LIN {X 0,Y 117.443,Z 618.499,A -85,B 0,C 180,E1 -30787.751,E2 -30787.751} C_VEL
LIN {X 0,Y 117.759,Z 615.991,A -85,B 0,C 180,E1 -30784.552,E2 -30784.552} C_VEL
LIN {X 0,Y 118.169,Z 614.006,A -85,B 0,C 180,E1 -30779.995,E2 -30779.995} C_VEL
LIN {X 0,Y 117.877,Z 614.864,A -85,B 0,C 180,E1 -30779.723,E2 -30779.723} C_VEL
LIN {X 0,Y 113.586,Z 625.245,A -85,B 0,C 180,E1 -30779.502,E2 -30779.502} C_VEL
LIN {X 0,Y 107.189,Z 637.349,A -85,B 0,C 180,E1 -30779.105,E2 -30779.105} C_VEL
LIN {X 0,Y 99.299,Z 648.745,A -85,B 0,C 180,E1 -30778.609,E2 -30778.609} C_VEL
LIN {X 0,Y 93.168,Z 656.16,A -85,B 0,C 180,E1 -30778.155,E2 -30778.155} C_VEL
LIN {X 0,Y 84.423,Z 664.947,A -85,B 0,C 180,E1 -30777.39,E2 -30777.39} C_VEL
LIN {X 0,Y 77.444,Z 670.933,A -85,B 0,C 180,E1 -30776.591,E2 -30776.591} C_VEL
LIN {X 0,Y 68.748,Z 677.241,A -85,B 0,C 180,E1 -30775.357,E2 -30775.357} C_VEL
LIN {X 0,Y 59.764,Z 682.696,A -85,B 0,C 180,E1 -30773.548,E2 -30773.548} C_VEL
LIN {X 0,Y 49.831,Z 687.613,A -85,B 0,C 180,E1 -30770.836,E2 -30770.836} C_VEL
LIN {X 0,Y 39.702,Z 691.58,A -85,B 0,C 180,E1 -30766.802,E2 -30766.802} C_VEL
LIN {X 0,Y 29.884,Z 694.52,A -85,B 0,C 180,E1 -30760.167,E2 -30760.167} C_VEL
LIN {X 0,Y 23.763,Z 696.03,A -85,B 0,C 180,E1 -30752.531,E2 -30752.531} C_VEL
LIN {X 0,Y 14.258,Z 697.578,A -85,B 0,C 180,E1 -30719.533,E2 -30719.533} C_VEL
LIN {X 0,Y 12.869,Z 697.867,A -85,B 0,C 180,E1 -30690,E2 -30690} C_VEL
LIN {X 0,Y 18.308,Z 696.97,A -85,B 0,C 180,E1 -30639.849,E2 -30639.849} C_VEL
LIN {X 0,Y 23.763,Z 696.03,A -85,B 0,C 180,E1 -30627.469,E2 -30627.469} C_VEL
LIN {X 0,Y 36.383,Z 692.67,A -85,B 0,C 180,E1 -30615.024,E2 -30615.024} C_VEL
LIN {X 0,Y 46.428,Z 689.041,A -85,B 0,C 180,E1 -30610.286,E2 -30610.286} C_VEL
LIN {X 0,Y 56.667,Z 684.307,A -85,B 0,C 180,E1 -30607.176,E2 -30607.176} C_VEL
LIN {X 0,Y 65.281,Z 679.425,A -85,B 0,C 180,E1 -30605.243,E2 -30605.243} C_VEL
LIN {X 0,Y 73.96,Z 673.555,A -85,B 0,C 180,E1 -30603.851,E2 -30603.851} C_VEL
LIN {X 0,Y 80.93,Z 668.066,A -85,B 0,C 180,E1 -30602.978,E2 -30602.978} C_VEL
LIN {X 0,Y 89.665,Z 659.855,A -85,B 0,C 180,E1 -30602.083,E2 -30602.083} C_VEL
LIN {X 0,Y 96.67,Z 652.036,A -85,B 0,C 180,E1 -30601.557,E2 -30601.557} C_VEL
LIN {X 0,Y 102.804,Z 643.96,A -85,B 0,C 180,E1 -30601.142,E2 -30601.142} C_VEL
LIN {X 0,Y 108.944,Z 634.208,A -85,B 0,C 180,E1 -30600.823,E2 -30600.823} C_VEL
LIN {X 0,Y 114.036,Z 624.238,A -85,B 0,C 180,E1 -30600.507,E2 -30600.507} C_VEL
LIN {X 0,Y 117.877,Z 614.869,A -85,B 0,C 180,E1 -30600.322,E2 -30600.322} C_VEL
LIN {X 0,Y 118.172,Z 613.998,A -85,B 0,C 180,E1 -30600.005,E2 -30600.005} C_VEL
LIN {X 0,Y 117.763,Z 615.989,A -85,B 0,C 180,E1 -30595.422,E2 -30595.422} C_VEL
LIN {X 0,Y 117.614,Z 617.596,A -85,B 0,C 180,E1 -30593.142,E2 -30593.142} C_VEL
LIN {X 0,Y 117.105,Z 620.39,A -85,B 0,C 180,E1 -30590.506,E2 -30590.506} C_VEL
LIN {X 0,Y 116.14,Z 624.865,A -85,B 0,C 180,E1 -30587.601,E2 -30587.601} C_VEL
LIN {X 0,Y 115.107,Z 628.526,A -85,B 0,C 180,E1 -30585.87,E2 -30585.87} C_VEL
LIN {X 0,Y 111.487,Z 638.971,A -85,B 0,C 180,E1 -30581.01,E2 -30581.01} C_VEL
LIN {X 0,Y 108.455,Z 647.592,A -85,B 0,C 180,E1 -30576.115,E2 -30576.115} C_VEL
LIN {X 0,Y 106.01,Z 655.467,A -85,B 0,C 180,E1 -30570.569,E2 -30570.569} C_VEL
LIN {X 0,Y 104.558,Z 661.545,A -85,B 0,C 180,E1 -30565.542,E2 -30565.542} C_VEL
LIN {X 0,Y 103.809,Z 669.53,A -85,B 0,C 180,E1 -30557.398,E2 -30557.398} C_VEL
LIN {X 0,Y 104.443,Z 673.875,A -85,B 0,C 180,E1 -30552.262,E2 -30552.262} C_VEL
LIN {X 0,Y 106.959,Z 679.238,A -85,B 0,C 180,E1 -30544.795,E2 -30544.795} C_VEL
LIN {X 0,Y 112.881,Z 684.586,A -85,B 0,C 180,E1 -30535.837,E2 -30535.837} C_VEL
LIN {X 0,Y 119.382,Z 687.768,A -85,B 0,C 180,E1 -30529.642,E2 -30529.642} C_VEL
LIN {X 0,Y 130.255,Z 690.725,A -85,B 0,C 180,E1 -30522.464,E2 -30522.464} C_VEL
LIN {X 0,Y 141.656,Z 692.301,A -85,B 0,C 180,E1 -30517.174,E2 -30517.174} C_VEL
LIN {X 0,Y 154.94,Z 692.973,A -85,B 0,C 180,E1 -30512.6,E2 -30512.6} C_VEL
LIN {X 0,Y 164.279,Z 692.971,A -85,B 0,C 180,E1 -30510,E2 -30510} C_VEL
LIN {X 0,Y 146.004,Z 692.638,A -85,B 0,C 180,E1 -30504.476,E2 -30504.476} C_VEL
LIN {X 0,Y 144.157,Z 692.496,A -85,B 0,C 180,E1 -30503.795,E2 -30503.795} C_VEL
LIN {X 0,Y 139.501,Z 692.247,A -85,B 0,C 180,E1 -30502.329,E2 -30502.329} C_VEL
LIN {X 0,Y 124.191,Z 691.562,A -85,B 0,C 180,E1 -30498.362,E2 -30498.362} C_VEL
LIN {X 0,Y 119.811,Z 691.066,A -85,B 0,C 180,E1 -30496.531,E2 -30496.531} C_VEL
LIN {X 0,Y 118.583,Z 690.851,A -85,B 0,C 180,E1 -30495.803,E2 -30495.803} C_VEL
LIN {X 0,Y 108.043,Z 687.465,A -85,B 0,C 180,E1 -30487.028,E2 -30487.028} C_VEL
LIN {X 0,Y 102.213,Z 683.666,A -85,B 0,C 180,E1 -30479.228,E2 -30479.228} C_VEL
LIN {X 0,Y 98.445,Z 678.262,A -85,B 0,C 180,E1 -30470.021,E2 -30470.021} C_VEL
LIN {X 0,Y 97.481,Z 673.186,A -85,B 0,C 180,E1 -30462.695,E2 -30462.695} C_VEL
LIN {X 0,Y 98.282,Z 666.575,A -85,B 0,C 180,E1 -30454.887,E2 -30454.887} C_VEL
LIN {X 0,Y 100.458,Z 659.553,A -85,B 0,C 180,E1 -30448.17,E2 -30448.17} C_VEL
LIN {X 0,Y 103.759,Z 651.316,A -85,B 0,C 180,E1 -30441.863,E2 -30441.863} C_VEL
LIN {X 0,Y 107.51,Z 642.683,A -85,B 0,C 180,E1 -30436.593,E2 -30436.593} C_VEL
LIN {X 0,Y 111.381,Z 633.584,A -85,B 0,C 180,E1 -30432.125,E2 -30432.125} C_VEL
LIN {X 0,Y 112.591,Z 630.569,A -85,B 0,C 180,E1 -30430.787,E2 -30430.787} C_VEL
LIN {X 0,Y 113.778,Z 627.253,A -85,B 0,C 180,E1 -30428.772,E2 -30428.772} C_VEL
LIN {X 0,Y 114.375,Z 624.991,A -85,B 0,C 180,E1 -30427.054,E2 -30427.054} C_VEL
LIN {X 0,Y 114.764,Z 623.365,A -85,B 0,C 180,E1 -30425.265,E2 -30425.265} C_VEL
LIN {X 0,Y 115.055,Z 622.207,A -85,B 0,C 180,E1 -30423.497,E2 -30423.497} C_VEL
LIN {X 0,Y 114.2,Z 624.038,A -85,B 0,C 180,E1 -30423.094,E2 -30423.094} C_VEL
LIN {X 0,Y 109.077,Z 634.01,A -85,B 0,C 180,E1 -30422.945,E2 -30422.945} C_VEL
LIN {X 0,Y 102.907,Z 643.764,A -85,B 0,C 180,E1 -30422.804,E2 -30422.804} C_VEL
LIN {X 0,Y 94.975,Z 654.029,A -85,B 0,C 180,E1 -30422.61,E2 -30422.61} C_VEL
LIN {X 0,Y 86.161,Z 663.191,A -85,B 0,C 180,E1 -30422.294,E2 -30422.294} C_VEL
LIN {X 0,Y 77.348,Z 670.737,A -85,B 0,C 180,E1 -30421.861,E2 -30421.861} C_VEL
LIN {X 0,Y 68.54,Z 677.044,A -85,B 0,C 180,E1 -30421.302,E2 -30421.302} C_VEL
LIN {X 0,Y 59.739,Z 682.319,A -85,B 0,C 180,E1 -30420.452,E2 -30420.452} C_VEL
LIN {X 0,Y 49.202,Z 687.416,A -85,B 0,C 180,E1 -30419.067,E2 -30419.067} C_VEL
LIN {X 0,Y 38.701,Z 691.383,A -85,B 0,C 180,E1 -30417.149,E2 -30417.149} C_VEL
LIN {X 0,Y 28.273,Z 694.323,A -85,B 0,C 180,E1 -30413.877,E2 -30413.877} C_VEL
LIN {X 0,Y 21.426,Z 695.833,A -85,B 0,C 180,E1 -30409.747,E2 -30409.747} C_VEL
LIN {X 0,Y 8.799,Z 697.381,A -85,B 0,C 180,E1 -30383.004,E2 -30383.004} C_VEL
LIN {X 0,Y 5.756,Z 697.671,A -85,B 0,C 180,E1 -30330,E2 -30330} C_VEL
LIN {X 0,Y 14.791,Z 696.773,A -85,B 0,C 180,E1 -30258.136,E2 -30258.136} C_VEL
LIN {X 0,Y 21.426,Z 695.833,A -85,B 0,C 180,E1 -30250.252,E2 -30250.252} C_VEL
LIN {X 0,Y 35.216,Z 692.474,A -85,B 0,C 180,E1 -30243.768,E2 -30243.768} C_VEL
LIN {X 0,Y 45.697,Z 688.844,A -85,B 0,C 180,E1 -30241.474,E2 -30241.474} C_VEL
LIN {X 0,Y 55.645,Z 684.404,A -85,B 0,C 180,E1 -30240.011,E2 -30240.011} C_VEL
LIN {X 0,Y 66.779,Z 678.135,A -85,B 0,C 180,E1 -30238.818,E2 -30238.818} C_VEL
LIN {X 0,Y 75.588,Z 672.046,A -85,B 0,C 180,E1 -30238.197,E2 -30238.197} C_VEL
LIN {X 0,Y 82.636,Z 666.31,A -85,B 0,C 180,E1 -30237.856,E2 -30237.856} C_VEL
LIN {X 0,Y 89.688,Z 659.658,A -85,B 0,C 180,E1 -30237.543,E2 -30237.543} C_VEL
LIN {X 0,Y 96.738,Z 651.84,A -85,B 0,C 180,E1 -30237.347,E2 -30237.347} C_VEL
LIN {X 0,Y 102.907,Z 643.764,A -85,B 0,C 180,E1 -30237.192,E2 -30237.192} C_VEL
LIN {X 0,Y 109.074,Z 634.012,A -85,B 0,C 180,E1 -30237.087,E2 -30237.087} C_VEL
LIN {X 0,Y 114.222,Z 623.981,A -85,B 0,C 180,E1 -30236.941,E2 -30236.941} C_VEL
LIN {X 0,Y 114.7,Z 622.912,A -85,B 0,C 180,E1 -30236.943,E2 -30236.943} C_VEL
LIN {X 0,Y 115.069,Z 622.175,A -85,B 0,C 180,E1 -30236.504,E2 -30236.504} C_VEL
LIN {X 0,Y 114.776,Z 623.339,A -85,B 0,C 180,E1 -30234.735,E2 -30234.735} C_VEL
LIN {X 0,Y 114.111,Z 626.031,A -85,B 0,C 180,E1 -30232.084,E2 -30232.084} C_VEL
LIN {X 0,Y 113.261,Z 628.786,A -85,B 0,C 180,E1 -30230.225,E2 -30230.225} C_VEL
LIN {X 0,Y 111.785,Z 632.565,A -85,B 0,C 180,E1 -30228.324,E2 -30228.324} C_VEL
LIN {X 0,Y 108.15,Z 641.164,A -85,B 0,C 180,E1 -30224.221,E2 -30224.221} C_VEL
LIN {X 0,Y 104.826,Z 648.774,A -85,B 0,C 180,E1 -30219.82,E2 -30219.82} C_VEL
LIN {X 0,Y 102.329,Z 654.783,A -85,B 0,C 180,E1 -30215.671,E2 -30215.671} C_VEL
LIN {X 0,Y 99.693,Z 661.815,A -85,B 0,C 180,E1 -30209.833,E2 -30209.833} C_VEL
LIN {X 0,Y 97.787,Z 669.151,A -85,B 0,C 180,E1 -30202.238,E2 -30202.238} C_VEL
LIN {X 0,Y 97.688,Z 675.553,A -85,B 0,C 180,E1 -30194.002,E2 -30194.002} C_VEL
LIN {X 0,Y 99.545,Z 680.564,A -85,B 0,C 180,E1 -30186.239,E2 -30186.239} C_VEL
LIN {X 0,Y 103.704,Z 684.913,A -85,B 0,C 180,E1 -30178.25,E2 -30178.25} C_VEL
LIN {X 0,Y 108.04,Z 687.465,A -85,B 0,C 180,E1 -30172.973,E2 -30172.973} C_VEL
LIN {X 0,Y 116.689,Z 690.455,A -85,B 0,C 180,E1 -30165.517,E2 -30165.517} C_VEL
LIN {X 0,Y 128.026,Z 692.417,A -85,B 0,C 180,E1 -30158.879,E2 -30158.879} C_VEL
LIN {X 0,Y 143.096,Z 693.294,A -85,B 0,C 180,E1 -30152.815,E2 -30152.815} C_VEL
LIN {X 0,Y 152.364,Z 693.301,A -85,B 0,C 180,E1 -30150,E2 -30150} C_VEL
LIN {X 0,Y 139.359,Z 693.208,A -85,B 0,C 180,E1 -30145.887,E2 -30145.887} C_VEL
LIN {X 0,Y 126.564,Z 692.278,A -85,B 0,C 180,E1 -30140.411,E2 -30140.411} C_VEL
LIN {X 0,Y 118.583,Z 690.851,A -85,B 0,C 180,E1 -30135.803,E2 -30135.803} C_VEL
LIN {X 0,Y 114.711,Z 690.267,A -85,B 0,C 180,E1 -30133.626,E2 -30133.626} C_VEL
LIN {X 0,Y 101.783,Z 688.638,A -85,B 0,C 180,E1 -30127.171,E2 -30127.171} C_VEL
LIN {X 0,Y 98.483,Z 687.64,A -85,B 0,C 180,E1 -30124.443,E2 -30124.443} C_VEL
LIN {X 0,Y 97.672,Z 687.193,A -85,B 0,C 180,E1 -30123.431,E2 -30123.431} C_VEL
LIN {X 0,Y 93.554,Z 683.757,A -85,B 0,C 180,E1 -30115.713,E2 -30115.713} C_VEL
LIN {X 0,Y 91.224,Z 678.53,A -85,B 0,C 180,E1 -30106.103,E2 -30106.103} C_VEL
LIN {X 0,Y 91.415,Z 673.13,A -85,B 0,C 180,E1 -30097.946,E2 -30097.946} C_VEL
LIN {X 0,Y 93.272,Z 667.087,A -85,B 0,C 180,E1 -30090.562,E2 -30090.562} C_VEL
LIN {X 0,Y 96.531,Z 659.898,A -85,B 0,C 180,E1 -30083.595,E2 -30083.595} C_VEL
LIN {X 0,Y 100.499,Z 652.251,A -85,B 0,C 180,E1 -30077.733,E2 -30077.733} C_VEL
LIN {X 0,Y 104.974,Z 643.783,A -85,B 0,C 180,E1 -30072.617,E2 -30072.617} C_VEL
LIN {X 0,Y 109.775,Z 634.122,A -85,B 0,C 180,E1 -30067.933,E2 -30067.933} C_VEL
LIN {X 0,Y 110.243,Z 633.033,A -85,B 0,C 180,E1 -30067.319,E2 -30067.319} C_VEL
LIN {X 0,Y 109.186,Z 634.691,A -85,B 0,C 180,E1 -30066.667,E2 -30066.667} C_VEL
LIN {X 0,Y 101.734,Z 646.133,A -85,B 0,C 180,E1 -30066.763,E2 -30066.763} C_VEL
LIN {X 0,Y 93.796,Z 655.766,A -85,B 0,C 180,E1 -30066.885,E2 -30066.885} C_VEL
LIN {X 0,Y 84.975,Z 664.553,A -85,B 0,C 180,E1 -30067.035,E2 -30067.035} C_VEL
LIN {X 0,Y 77.907,Z 670.539,A -85,B 0,C 180,E1 -30067.115,E2 -30067.115} C_VEL
LIN {X 0,Y 69.072,Z 676.847,A -85,B 0,C 180,E1 -30067.231,E2 -30067.231} C_VEL
LIN {X 0,Y 60.223,Z 682.121,A -85,B 0,C 180,E1 -30067.28,E2 -30067.28} C_VEL
LIN {X 0,Y 49.602,Z 687.219,A -85,B 0,C 180,E1 -30067.337,E2 -30067.337} C_VEL
LIN {X 0,Y 39.005,Z 691.185,A -85,B 0,C 180,E1 -30067.697,E2 -30067.697} C_VEL
LIN {X 0,Y 28.409,Z 694.126,A -85,B 0,C 180,E1 -30068.301,E2 -30068.301} C_VEL
LIN {X 0,Y 21.345,Z 695.635,A -85,B 0,C 180,E1 -30068.978,E2 -30068.978} C_VEL
LIN {X 0,Y 7.264,Z 697.184,A -85,B 0,C 180,E1 -30074.645,E2 -30074.645} C_VEL
LIN {X 0,Y 1.343,Z 697.475,A -85,B 0,C 180,E1 -30150,E2 -30150} C_VEL
LIN {X 0,Y 14.283,Z 696.575,A -85,B 0,C 180,E1 -30229.759,E2 -30229.759} C_VEL
LIN {X 0,Y 21.345,Z 695.635,A -85,B 0,C 180,E1 -30231.022,E2 -30231.022} C_VEL
LIN {X 0,Y 35.466,Z 692.277,A -85,B 0,C 180,E1 -30232.216,E2 -30232.216} C_VEL
LIN {X 0,Y 46.066,Z 688.647,A -85,B 0,C 180,E1 -30232.59,E2 -30232.59} C_VEL
LIN {X 0,Y 56.684,Z 683.912,A -85,B 0,C 180,E1 -30232.692,E2 -30232.692} C_VEL
LIN {X 0,Y 67.305,Z 677.938,A -85,B 0,C 180,E1 -30232.739,E2 -30232.739} C_VEL
LIN {X 0,Y 76.144,Z 671.849,A -85,B 0,C 180,E1 -30232.837,E2 -30232.837} C_VEL
LIN {X 0,Y 83.206,Z 666.113,A -85,B 0,C 180,E1 -30232.957,E2 -30232.957} C_VEL
LIN {X 0,Y 90.272,Z 659.462,A -85,B 0,C 180,E1 -30233.038,E2 -30233.038} C_VEL
LIN {X 0,Y 97.324,Z 651.644,A -85,B 0,C 180,E1 -30233.171,E2 -30233.171} C_VEL
LIN {X 0,Y 103.497,Z 643.568,A -85,B 0,C 180,E1 -30233.268,E2 -30233.268} C_VEL
LIN {X 0,Y 109.17,Z 634.704,A -85,B 0,C 180,E1 -30233.38,E2 -30233.38} C_VEL
LIN {X 0,Y 110.22,Z 633.075,A -85,B 0,C 180,E1 -30232.679,E2 -30232.679} C_VEL
LIN {X 0,Y 107.201,Z 639.436,A -85,B 0,C 180,E1 -30229.539,E2 -30229.539} C_VEL
LIN {X 0,Y 102.878,Z 647.758,A -85,B 0,C 180,E1 -30225.104,E2 -30225.104} C_VEL
LIN {X 0,Y 99.152,Z 654.795,A -85,B 0,C 180,E1 -30220.508,E2 -30220.508} C_VEL
LIN {X 0,Y 95.086,Z 662.884,A -85,B 0,C 180,E1 -30213.682,E2 -30213.682} C_VEL
LIN {X 0,Y 92.412,Z 669.407,A -85,B 0,C 180,E1 -30206.777,E2 -30206.777} C_VEL
LIN {X 0,Y 91.145,Z 675.365,A -85,B 0,C 180,E1 -30198.846,E2 -30198.846} C_VEL
LIN {X 0,Y 91.811,Z 680.718,A -85,B 0,C 180,E1 -30190.061,E2 -30190.061} C_VEL
LIN {X 0,Y 94.843,Z 685.153,A -85,B 0,C 180,E1 -30181.245,E2 -30181.245} C_VEL
LIN {X 0,Y 99.773,Z 688.355,A -85,B 0,C 180,E1 -30173.709,E2 -30173.709} C_VEL
LIN {X 0,Y 109.071,Z 691.344,A -85,B 0,C 180,E1 -30164.891,E2 -30164.891} C_VEL
LIN {X 0,Y 115.719,Z 692.583,A -85,B 0,C 180,E1 -30160.498,E2 -30160.498} C_VEL
LIN {X 0,Y 126.949,Z 693.553,A -85,B 0,C 180,E1 -30154.865,E2 -30154.865} C_VEL
LIN {X 0,Y 140.481,Z 693.629,A -85,B 0,C 180,E1 -30150,E2 -30150} C_VEL
LIN {X 0,Y 126.947,Z 693.555,A -85,B 0,C 180,E1 -30145.143,E2 -30145.143} C_VEL
LIN {X 0,Y 112.941,Z 692.113,A -85,B 0,C 180,E1 -30137.816,E2 -30137.816} C_VEL
LIN {X 0,Y 103.287,Z 689.725,A -85,B 0,C 180,E1 -30130.11,E2 -30130.11} C_VEL
LIN {X 0,Y 97.672,Z 687.193,A -85,B 0,C 180,E1 -30123.431,E2 -30123.431} C_VEL
LIN {X 0,Y 95.079,Z 686.008,A -85,B 0,C 180,E1 -30120.357,E2 -30120.357} C_VEL
LIN {X 0,Y 86.327,Z 683.064,A -85,B 0,C 180,E1 -30110.705,E2 -30110.705} C_VEL
LIN {X 0,Y 84.792,Z 681.6,A -85,B 0,C 180,E1 -30107.025,E2 -30107.025} C_VEL
LIN {X 0,Y 84.618,Z 681.014,A -85,B 0,C 180,E1 -30105.764,E2 -30105.764} C_VEL
LIN {X 0,Y 85.582,Z 674.635,A -85,B 0,C 180,E1 -30094.795,E2 -30094.795} C_VEL
LIN {X 0,Y 89.365,Z 666.65,A -85,B 0,C 180,E1 -30084.808,E2 -30084.808} C_VEL
LIN {X 0,Y 93.127,Z 660.513,A -85,B 0,C 180,E1 -30078.914,E2 -30078.914} C_VEL
LIN {X 0,Y 98.879,Z 651.385,A -85,B 0,C 180,E1 -30072.233,E2 -30072.233} C_VEL
LIN {X 0,Y 100.176,Z 649.253,A -85,B 0,C 180,E1 -30070.833,E2 -30070.833} C_VEL
LIN {X 0,Y 93.159,Z 657.418,A -85,B 0,C 180,E1 -30071.269,E2 -30071.269} C_VEL
LIN {X 0,Y 86.138,Z 664.356,A -85,B 0,C 180,E1 -30071.743,E2 -30071.743} C_VEL
LIN {X 0,Y 79.106,Z 670.343,A -85,B 0,C 180,E1 -30072.241,E2 -30072.241} C_VEL
LIN {X 0,Y 70.324,Z 676.65,A -85,B 0,C 180,E1 -30072.999,E2 -30072.999} C_VEL
LIN {X 0,Y 61.537,Z 681.924,A -85,B 0,C 180,E1 -30073.892,E2 -30073.892} C_VEL
LIN {X 0,Y 51.01,Z 687.021,A -85,B 0,C 180,E1 -30075.327,E2 -30075.327} C_VEL
LIN {X 0,Y 40.584,Z 690.988,A -85,B 0,C 180,E1 -30077.742,E2 -30077.742} C_VEL
LIN {X 0,Y 30.266,Z 693.93,A -85,B 0,C 180,E1 -30081.747,E2 -30081.747} C_VEL
LIN {X 0,Y 23.541,Z 695.438,A -85,B 0,C 180,E1 -30086.414,E2 -30086.414} C_VEL
LIN {X 0,Y 11.387,Z 696.987,A -85,B 0,C 180,E1 -30111.89,E2 -30111.89} C_VEL
LIN {X 0,Y 8.433,Z 697.279,A -85,B 0,C 180,E1 -30150,E2 -30150} C_VEL
LIN {X 0,Y 17.064,Z 696.378,A -85,B 0,C 180,E1 -30205.457,E2 -30205.457} C_VEL
LIN {X 0,Y 23.542,Z 695.438,A -85,B 0,C 180,E1 -30213.585,E2 -30213.585} C_VEL
LIN {X 0,Y 37.113,Z 692.08,A -85,B 0,C 180,E1 -30221.231,E2 -30221.231} C_VEL
LIN {X 0,Y 47.511,Z 688.451,A -85,B 0,C 180,E1 -30224.047,E2 -30224.047} C_VEL
LIN {X 0,Y 55.616,Z 684.943,A -85,B 0,C 180,E1 -30225.372,E2 -30225.372} C_VEL
LIN {X 0,Y 66.815,Z 678.834,A -85,B 0,C 180,E1 -30226.646,E2 -30226.646} C_VEL
LIN {X 0,Y 75.601,Z 672.963,A -85,B 0,C 180,E1 -30227.443,E2 -30227.443} C_VEL
LIN {X 0,Y 82.618,Z 667.476,A -85,B 0,C 180,E1 -30228.03,E2 -30228.03} C_VEL
LIN {X 0,Y 91.409,Z 659.265,A -85,B 0,C 180,E1 -30228.602,E2 -30228.602} C_VEL
LIN {X 0,Y 98.422,Z 651.447,A -85,B 0,C 180,E1 -30229.061,E2 -30229.061} C_VEL
LIN {X 0,Y 100.213,Z 649.247,A -85,B 0,C 180,E1 -30229.057,E2 -30229.057} C_VEL
LIN {X 0,Y 95.856,Z 656.134,A -85,B 0,C 180,E1 -30224.553,E2 -30224.553} C_VEL
LIN {X 0,Y 90.993,Z 663.897,A -85,B 0,C 180,E1 -30217.947,E2 -30217.947} C_VEL
LIN {X 0,Y 87.501,Z 670.11,A -85,B 0,C 180,E1 -30211.198,E2 -30211.198} C_VEL
LIN {X 0,Y 85.508,Z 674.843,A -85,B 0,C 180,E1 -30204.886,E2 -30204.886} C_VEL
LIN {X 0,Y 84.56,Z 680.62,A -85,B 0,C 180,E1 -30195.064,E2 -30195.064} C_VEL
LIN {X 0,Y 86.454,Z 685.429,A -85,B 0,C 180,E1 -30184.683,E2 -30184.683} C_VEL
LIN {X 0,Y 89.357,Z 688.037,A -85,B 0,C 180,E1 -30178.158,E2 -30178.158} C_VEL
LIN {X 0,Y 96.479,Z 691.081,A -85,B 0,C 180,E1 -30168.762,E2 -30168.762} C_VEL
LIN {X 0,Y 107.096,Z 693.104,A -85,B 0,C 180,E1 -30160.186,E2 -30160.186} C_VEL
LIN {X 0,Y 120.064,Z 693.922,A -85,B 0,C 180,E1 -30153.356,E2 -30153.356} C_VEL
LIN {X 0,Y 128.809,Z 693.952,A -85,B 0,C 180,E1 -30150,E2 -30150} C_VEL
LIN {X 0,Y 113.19,Z 693.668,A -85,B 0,C 180,E1 -30143.383,E2 -30143.383} C_VEL
LIN {X 0,Y 104.921,Z 692.887,A -85,B 0,C 180,E1 -30138.408,E2 -30138.408} C_VEL
LIN {X 0,Y 96.479,Z 691.081,A -85,B 0,C 180,E1 -30131.237,E2 -30131.237} C_VEL
LIN {X 0,Y 88.743,Z 687.517,A -85,B 0,C 180,E1 -30120.577,E2 -30120.577} C_VEL
LIN {X 0,Y 85.418,Z 683.748,A -85,B 0,C 180,E1 -30111.394,E2 -30111.394} C_VEL
LIN {X 0,Y 84.618,Z 681.014,A -85,B 0,C 180,E1 -30105.764,E2 -30105.764} C_VEL
LIN {X 0,Y 83.985,Z 679.338,A -85,B 0,C 180,E1 -30101.931,E2 -30101.931} C_VEL
LIN {X 0,Y 81.448,Z 674.737,A -85,B 0,C 180,E1 -30090.111,E2 -30090.111} C_VEL
LIN {X 0,Y 82.048,Z 672.59,A -85,B 0,C 180,E1 -30086.297,E2 -30086.297} C_VEL
LIN {X 0,Y 82.552,Z 671.741,A -85,B 0,C 180,E1 -30085.118,E2 -30085.118} C_VEL
LIN {X 0,Y 86.635,Z 666.009,A -85,B 0,C 180,E1 -30078.505,E2 -30078.505} C_VEL
LIN {X 0,Y 88.039,Z 664.143,A -85,B 0,C 180,E1 -30076.678,E2 -30076.678} C_VEL
LIN {X 0,Y 87.861,Z 664.16,A -85,B 0,C 180,E1 -30076.288,E2 -30076.288} C_VEL
LIN {X 0,Y 80.914,Z 670.146,A -85,B 0,C 180,E1 -30077.173,E2 -30077.173} C_VEL
LIN {X 0,Y 72.266,Z 676.453,A -85,B 0,C 180,E1 -30078.522,E2 -30078.522} C_VEL
LIN {X 0,Y 63.633,Z 681.726,A -85,B 0,C 180,E1 -30080.152,E2 -30080.152} C_VEL
LIN {X 0,Y 53.345,Z 686.824,A -85,B 0,C 180,E1 -30082.748,E2 -30082.748} C_VEL
LIN {X 0,Y 43.294,Z 690.79,A -85,B 0,C 180,E1 -30086.77,E2 -30086.77} C_VEL
LIN {X 0,Y 33.556,Z 693.733,A -85,B 0,C 180,E1 -30093.097,E2 -30093.097} C_VEL
LIN {X 0,Y 27.471,Z 695.24,A -85,B 0,C 180,E1 -30099.872,E2 -30099.872} C_VEL
LIN {X 0,Y 17.543,Z 696.791,A -85,B 0,C 180,E1 -30126.384,E2 -30126.384} C_VEL
LIN {X 0,Y 15.542,Z 697.082,A -85,B 0,C 180,E1 -30150,E2 -30150} C_VEL
LIN {X 0,Y 21.908,Z 696.181,A -85,B 0,C 180,E1 -30189.911,E2 -30189.911} C_VEL
LIN {X 0,Y 27.471,Z 695.24,A -85,B 0,C 180,E1 -30200.128,E2 -30200.128} C_VEL
LIN {X 0,Y 39.991,Z 691.882,A -85,B 0,C 180,E1 -30211.484,E2 -30211.484} C_VEL
LIN {X 0,Y 49.949,Z 688.253,A -85,B 0,C 180,E1 -30216.144,E2 -30216.144} C_VEL
LIN {X 0,Y 60.19,Z 683.517,A -85,B 0,C 180,E1 -30219.083,E2 -30219.083} C_VEL
LIN {X 0,Y 70.537,Z 677.545,A -85,B 0,C 180,E1 -30221.178,E2 -30221.178} C_VEL
LIN {X 0,Y 79.19,Z 671.456,A -85,B 0,C 180,E1 -30222.561,E2 -30222.561} C_VEL
LIN {X 0,Y 85.714,Z 666.088,A -85,B 0,C 180,E1 -30223.449,E2 -30223.449} C_VEL
LIN {X 0,Y 87.862,Z 664.16,A -85,B 0,C 180,E1 -30223.712,E2 -30223.712} C_VEL
LIN {X 0,Y 88.039,Z 664.143,A -85,B 0,C 180,E1 -30223.321,E2 -30223.321} C_VEL
LIN {X 0,Y 83.847,Z 669.909,A -85,B 0,C 180,E1 -30217.22,E2 -30217.22} C_VEL
LIN {X 0,Y 79.779,Z 676.411,A -85,B 0,C 180,E1 -30208.102,E2 -30208.102} C_VEL
LIN {X 0,Y 78.039,Z 681.486,A -85,B 0,C 180,E1 -30198.662,E2 -30198.662} C_VEL
LIN {X 0,Y 78.573,Z 685.701,A -85,B 0,C 180,E1 -30188.764,E2 -30188.764} C_VEL
LIN {X 0,Y 81.215,Z 688.752,A -85,B 0,C 180,E1 -30180.093,E2 -30180.093} C_VEL
LIN {X 0,Y 84.533,Z 690.555,A -85,B 0,C 180,E1 -30173.881,E2 -30173.881} C_VEL
LIN {X 0,Y 94.469,Z 693.182,A -85,B 0,C 180,E1 -30162.896,E2 -30162.896} C_VEL
LIN {X 0,Y 108.891,Z 694.232,A -85,B 0,C 180,E1 -30153.7,E2 -30153.7} C_VEL
LIN {X 0,Y 117.313,Z 694.269,A -85,B 0,C 180,E1 -30150,E2 -30150} C_VEL
LIN {X 0,Y 105.853,Z 694.207,A -85,B 0,C 180,E1 -30144.741,E2 -30144.741} C_VEL
LIN {X 0,Y 93.894,Z 693.094,A -85,B 0,C 180,E1 -30136.638,E2 -30136.638} C_VEL
LIN {X 0,Y 84.059,Z 690.299,A -85,B 0,C 180,E1 -30125.289,E2 -30125.289} C_VEL
LIN {X 0,Y 80.697,Z 688.313,A -85,B 0,C 180,E1 -30118.497,E2 -30118.497} C_VEL
LIN {X 0,Y 77.969,Z 683.667,A -85,B 0,C 180,E1 -30106.133,E2 -30106.133} C_VEL
LIN {X 0,Y 78.844,Z 678.402,A -85,B 0,C 180,E1 -30095.283,E2 -30095.283} C_VEL
LIN {X 0,Y 81.805,Z 672.898,A -85,B 0,C 180,E1 -30086.628,E2 -30086.628} C_VEL
LIN {X 0,Y 82.552,Z 671.741,A -85,B 0,C 180,E1 -30085.118,E2 -30085.118} C_VEL
LIN {X 0,Y 82.231,Z 671.692,A -85,B 0,C 180,E1 -30084.439,E2 -30084.439} C_VEL
LIN {X 0,Y 80.572,Z 672.563,A -85,B 0,C 180,E1 -30083.685,E2 -30083.685} C_VEL
LIN {X 0,Y 77.536,Z 674.534,A -85,B 0,C 180,E1 -30083.409,E2 -30083.409} C_VEL
LIN {X 0,Y 70.473,Z 679.098,A -85,B 0,C 180,E1 -30084.753,E2 -30084.753} C_VEL
LIN {X 0,Y 64.348,Z 682.64,A -85,B 0,C 180,E1 -30086.557,E2 -30086.557} C_VEL
LIN {X 0,Y 56.486,Z 686.627,A -85,B 0,C 180,E1 -30089.433,E2 -30089.433} C_VEL
LIN {X 0,Y 46.936,Z 690.594,A -85,B 0,C 180,E1 -30094.559,E2 -30094.559} C_VEL
LIN {X 0,Y 37.929,Z 693.536,A -85,B 0,C 180,E1 -30102.169,E2 -30102.169} C_VEL
LIN {X 0,Y 32.51,Z 695.043,A -85,B 0,C 180,E1 -30109.569,E2 -30109.569} C_VEL
LIN {X 0,Y 24.25,Z 696.593,A -85,B 0,C 180,E1 -30133.154,E2 -30133.154} C_VEL
LIN {X 0,Y 22.64,Z 696.886,A -85,B 0,C 180,E1 -30150,E2 -30150} C_VEL
LIN {X 0,Y 27.749,Z 695.984,A -85,B 0,C 180,E1 -30180.433,E2 -30180.433} C_VEL
LIN {X 0,Y 32.51,Z 695.043,A -85,B 0,C 180,E1 -30190.431,E2 -30190.431} C_VEL
LIN {X 0,Y 43.855,Z 691.685,A -85,B 0,C 180,E1 -30203.252,E2 -30203.252} C_VEL
LIN {X 0,Y 53.239,Z 688.056,A -85,B 0,C 180,E1 -30209.099,E2 -30209.099} C_VEL
LIN {X 0,Y 61.066,Z 684.41,A -85,B 0,C 180,E1 -30212.334,E2 -30212.334} C_VEL
LIN {X 0,Y 71.598,Z 678.351,A -85,B 0,C 180,E1 -30215.5,E2 -30215.5} C_VEL
LIN {X 0,Y 76.518,Z 675.149,A -85,B 0,C 180,E1 -30216.703,E2 -30216.703} C_VEL
LIN {X 0,Y 72.132,Z 681.778,A -85,B 0,C 180,E1 -30204.236,E2 -30204.236} C_VEL
LIN {X 0,Y 71.225,Z 685.97,A -85,B 0,C 180,E1 -30193.686,E2 -30193.686} C_VEL
LIN {X 0,Y 72.377,Z 688.588,A -85,B 0,C 180,E1 -30185.634,E2 -30185.634} C_VEL
LIN {X 0,Y 76.926,Z 691.599,A -85,B 0,C 180,E1 -30174.013,E2 -30174.013} C_VEL
LIN {X 0,Y 86.343,Z 693.736,A -85,B 0,C 180,E1 -30162.415,E2 -30162.415} C_VEL
LIN {X 0,Y 98.59,Z 694.541,A -85,B 0,C 180,E1 -30153.742,E2 -30153.742} C_VEL
LIN {X 0,Y 106.034,Z 694.581,A -85,B 0,C 180,E1 -30150,E2 -30150} C_VEL
LIN {X 0,Y 90.5,Z 694.175,A -85,B 0,C 180,E1 -30141.065,E2 -30141.065} C_VEL
LIN {X 0,Y 81.208,Z 692.798,A -85,B 0,C 180,E1 -30132.144,E2 -30132.144} C_VEL
LIN {X 0,Y 74.962,Z 690.58,A -85,B 0,C 180,E1 -30122.046,E2 -30122.046} C_VEL
LIN {X 0,Y 71.771,Z 687.685,A -85,B 0,C 180,E1 -30111.556,E2 -30111.556} C_VEL
LIN {X 0,Y 71.375,Z 683.795,A -85,B 0,C 180,E1 -30100.444,E2 -30100.444} C_VEL
LIN {X 0,Y 73.457,Z 679.315,A -85,B 0,C 180,E1 -30090.564,E2 -30090.564} C_VEL
LIN {X 0,Y 76.514,Z 675.149,A -85,B 0,C 180,E1 -30083.291,E2 -30083.291} C_VEL
LIN {X 0,Y 66.422,Z 681.529,A -85,B 0,C 180,E1 -30085.926,E2 -30085.926} C_VEL
LIN {X 0,Y 64.348,Z 682.64,A -85,B 0,C 180,E1 -30086.557,E2 -30086.557} C_VEL
LIN {X 0,Y 59.633,Z 685.332,A -85,B 0,C 180,E1 -30088.872,E2 -30088.872} C_VEL
LIN {X 0,Y 50.567,Z 690.208,A -85,B 0,C 180,E1 -30098.632,E2 -30098.632} C_VEL
LIN {X 0,Y 45.747,Z 692.463,A -85,B 0,C 180,E1 -30105.643,E2 -30105.643} C_VEL
LIN {X 0,Y 43.097,Z 693.32,A -85,B 0,C 180,E1 -30109.161,E2 -30109.161} C_VEL
LIN {X 0,Y 38.223,Z 694.846,A -85,B 0,C 180,E1 -30116.523,E2 -30116.523} C_VEL
LIN {X 0,Y 31.137,Z 696.396,A -85,B 0,C 180,E1 -30136.956,E2 -30136.956} C_VEL
LIN {X 0,Y 29.755,Z 696.689,A -85,B 0,C 180,E1 -30150,E2 -30150} C_VEL
LIN {X 0,Y 34.093,Z 695.787,A -85,B 0,C 180,E1 -30174.348,E2 -30174.348} C_VEL
LIN {X 0,Y 38.223,Z 694.846,A -85,B 0,C 180,E1 -30183.477,E2 -30183.477} C_VEL
LIN {X 0,Y 48.467,Z 691.487,A -85,B 0,C 180,E1 -30196.471,E2 -30196.471} C_VEL
LIN {X 0,Y 57.231,Z 687.859,A -85,B 0,C 180,E1 -30202.958,E2 -30202.958} C_VEL
LIN {X 0,Y 61.868,Z 685.724,A -85,B 0,C 180,E1 -30205.403,E2 -30205.403} C_VEL
LIN {X 0,Y 65.716,Z 684.005,A -85,B 0,C 180,E1 -30205.907,E2 -30205.907} C_VEL
LIN {X 0,Y 64.669,Z 688.92,A -85,B 0,C 180,E1 -30190.487,E2 -30190.487} C_VEL
LIN {X 0,Y 66.251,Z 690.88,A -85,B 0,C 180,E1 -30181.953,E2 -30181.953} C_VEL
LIN {X 0,Y 74.133,Z 693.763,A -85,B 0,C 180,E1 -30166.523,E2 -30166.523} C_VEL
LIN {X 0,Y 87.084,Z 694.836,A -85,B 0,C 180,E1 -30154.629,E2 -30154.629} C_VEL
LIN {X 0,Y 94.956,Z 694.887,A -85,B 0,C 180,E1 -30150,E2 -30150} C_VEL
LIN {X 0,Y 84.815,Z 694.815,A -85,B 0,C 180,E1 -30143.832,E2 -30143.832} C_VEL
LIN {X 0,Y 73.585,Z 693.649,A -85,B 0,C 180,E1 -30132.731,E2 -30132.731} C_VEL
LIN {X 0,Y 66.292,Z 690.856,A -85,B 0,C 180,E1 -30117.99,E2 -30117.99} C_VEL
LIN {X 0,Y 64.647,Z 688.86,A -85,B 0,C 180,E1 -30109.287,E2 -30109.287} C_VEL
LIN {X 0,Y 65.625,Z 684.057,A -85,B 0,C 180,E1 -30094.134,E2 -30094.134} C_VEL
LIN {X 0,Y 62.387,Z 685.459,A -85,B 0,C 180,E1 -30094.269,E2 -30094.269} C_VEL
LIN {X 0,Y 54.21,Z 689.273,A -85,B 0,C 180,E1 -30098.936,E2 -30098.936} C_VEL
LIN {X 0,Y 43.097,Z 693.32,A -85,B 0,C 180,E1 -30109.161,E2 -30109.161} C_VEL
LIN {X 0,Y 39.512,Z 694.631,A -85,B 0,C 180,E1 -30115.422,E2 -30115.422} C_VEL
LIN {X 0,Y 37.222,Z 695.575,A -85,B 0,C 180,E1 -30123.482,E2 -30123.482} C_VEL
LIN {X 0,Y 36.206,Z 696.454,A -85,B 0,C 180,E1 -30142.128,E2 -30142.128} C_VEL
LIN {X 0,Y 37.226,Z 696.37,A -85,B 0,C 180,E1 -30154.521,E2 -30154.521} C_VEL
LIN {X 0,Y 40.693,Z 695.59,A -85,B 0,C 180,E1 -30170.207,E2 -30170.207} C_VEL
LIN {X 0,Y 44.347,Z 694.649,A -85,B 0,C 180,E1 -30178.387,E2 -30178.387} C_VEL
LIN {X 0,Y 53.631,Z 691.29,A -85,B 0,C 180,E1 -30190.935,E2 -30190.935} C_VEL
LIN {X 0,Y 57.598,Z 689.982,A -85,B 0,C 180,E1 -30192.953,E2 -30192.953} C_VEL
LIN {X 0,Y 58.832,Z 691.924,A -85,B 0,C 180,E1 -30183.278,E2 -30183.278} C_VEL
LIN {X 0,Y 65.971,Z 694.29,A -85,B 0,C 180,E1 -30166.544,E2 -30166.544} C_VEL
LIN {X 0,Y 76.413,Z 695.132,A -85,B 0,C 180,E1 -30155.277,E2 -30155.277} C_VEL
LIN {X 0,Y 84.029,Z 695.189,A -85,B 0,C 180,E1 -30150,E2 -30150} C_VEL
LIN {X 0,Y 69.789,Z 694.756,A -85,B 0,C 180,E1 -30138.381,E2 -30138.381} C_VEL
LIN {X 0,Y 64.399,Z 694.045,A -85,B 0,C 180,E1 -30130.889,E2 -30130.889} C_VEL
LIN {X 0,Y 58.842,Z 691.919,A -85,B 0,C 180,E1 -30116.707,E2 -30116.707} C_VEL
LIN {X 0,Y 57.616,Z 689.974,A -85,B 0,C 180,E1 -30107.028,E2 -30107.028} C_VEL
LIN {X 0,Y 53.632,Z 691.29,A -85,B 0,C 180,E1 -30109.065,E2 -30109.065} C_VEL
LIN {X 0,Y 44.347,Z 694.649,A -85,B 0,C 180,E1 -30121.613,E2 -30121.613} C_VEL
LIN {X 0,Y 38.104,Z 696.2,A -85,B 0,C 180,E1 -30139.371,E2 -30139.371} C_VEL
LIN {X 0,Y 36.859,Z 696.493,A -85,B 0,C 180,E1 -30150,E2 -30150} C_VEL
LIN {X 0,Y 37.226,Z 696.37,A -85,B 0,C 180,E1 -30154.521,E2 -30154.521} C_VEL
LIN {X 0,Y 39.242,Z 696.13,A -85,B 0,C 180,E1 -30161.817,E2 -30161.817} C_VEL
LIN {X 0,Y 42.797,Z 695.719,A -85,B 0,C 180,E1 -30167.34,E2 -30167.34} C_VEL
LIN {X 0,Y 51.464,Z 694.272,A -85,B 0,C 180,E1 -30175.188,E2 -30175.188} C_VEL
LIN {X 0,Y 53.356,Z 693.816,A -85,B 0,C 180,E1 -30176.709,E2 -30176.709} C_VEL
LIN {X 0,Y 59.675,Z 695.043,A -85,B 0,C 180,E1 -30163.624,E2 -30163.624} C_VEL
LIN {X 0,Y 70.323,Z 695.475,A -85,B 0,C 180,E1 -30152.251,E2 -30152.251} C_VEL
LIN {X 0,Y 73.261,Z 695.487,A -85,B 0,C 180,E1 -30150,E2 -30150} C_VEL
LIN {X 0,Y 63.901,Z 695.396,A -85,B 0,C 180,E1 -30141.754,E2 -30141.754} C_VEL
LIN {X 0,Y 54.124,Z 694.075,A -85,B 0,C 180,E1 -30125.332,E2 -30125.332} C_VEL
LIN {X 0,Y 53.379,Z 693.805,A -85,B 0,C 180,E1 -30123.24,E2 -30123.24} C_VEL
LIN {X 0,Y 50.729,Z 694.452,A -85,B 0,C 180,E1 -30125.442,E2 -30125.442} C_VEL
LIN {X 0,Y 45.109,Z 696.003,A -85,B 0,C 180,E1 -30141.037,E2 -30141.037} C_VEL
LIN {X 0,Y 43.955,Z 696.297,A -85,B 0,C 180,E1 -30150,E2 -30150} C_VEL
LIN {X 0,Y 47.465,Z 695.392,A -85,B 0,C 180,E1 -30167.225,E2 -30167.225} C_VEL
LIN {X 0,Y 50.729,Z 694.452,A -85,B 0,C 180,E1 -30174.558,E2 -30174.558} C_VEL
LIN {X 0,Y 51.464,Z 694.272,A -85,B 0,C 180,E1 -30175.188,E2 -30175.188} C_VEL
LIN {X 0,Y 52.383,Z 694.218,A -85,B 0,C 180,E1 -30175.012,E2 -30175.012} C_VEL
LIN {X 0,Y 53.517,Z 694.367,A -85,B 0,C 180,E1 -30173.206,E2 -30173.206} C_VEL
LIN {X 0,Y 54.428,Z 694.821,A -85,B 0,C 180,E1 -30168.361,E2 -30168.361} C_VEL
LIN {X 0,Y 55.711,Z 695.68,A -85,B 0,C 180,E1 -30158.835,E2 -30158.835} C_VEL
LIN {X 0,Y 57.792,Z 695.738,A -85,B 0,C 180,E1 -30154.771,E2 -30154.771} C_VEL
LIN {X 0,Y 58.384,Z 695.74,A -85,B 0,C 180,E1 -30154.094,E2 -30154.094} C_VEL
LIN {X 0,Y 62.776,Z 695.777,A -85,B 0,C 180,E1 -30150,E2 -30150} C_VEL
LIN {X 0,Y 54.153,Z 695.687,A -85,B 0,C 180,E1 -30140.78,E2 -30140.78} C_VEL
LIN {X 0,Y 52.175,Z 695.806,A -85,B 0,C 180,E1 -30142.259,E2 -30142.259} C_VEL
LIN {X 0,Y 51.078,Z 696.1,A -85,B 0,C 180,E1 -30150,E2 -30150} C_VEL
LIN {X 0,Y 52.198,Z 695.805,A -85,B 0,C 180,E1 -30157.738,E2 -30157.738} C_VEL
LIN {X 0,Y 54.143,Z 695.689,A -85,B 0,C 180,E1 -30159.179,E2 -30159.179} C_VEL
LIN {X 0,Y 58.384,Z 695.74,A -85,B 0,C 180,E1 -30154.094,E2 -30154.094} C_VEL
LIN {X 0,Y 58.384,Z 695.74,A -85,B 0,C 180,E1 -30154.094,E2 -30154.094}

QRS_NEXT_CUT()

QRS_NEXT()
QRS_HOME()

END
